SUBAPPLICATION Uebung_087a2_AX (* Beispiel für E_DEMUX_4, mit Plug and Socket *)
  (* Standard: 61499-2; Description: Copyright (c) 2026 Meisterschulen am Ostbahnhof This program and the accompanying materials are made available under the terms of the Eclipse Public License 2.0 which is available at https://www.eclipse.org/legal/epl-2.0/ SPDX-License-Identifier: EPL-2.0 *)
  (* Version 1.0, 2026-09-10, Franz Höpfinger, Meisterschulen am Ostbahnhof, initial API and implementation and/or initial documentation *)
  PACKAGE Uebungen;
  IMPORT logiBUS::io::DI::logiBUS_DI::Input_I1;
  IMPORT logiBUS::io::DI::logiBUS_DI::Input_I2;
  IMPORT logiBUS::io::DI::logiBUS_DI::Input_I3;
  IMPORT logiBUS::io::DI::logiBUS_DI::Input_I4;
  IMPORT logiBUS::io::DQ::logiBUS_DO::Output_Q1;
  IMPORT logiBUS::io::DQ::logiBUS_DO::Output_Q2;
  IMPORT logiBUS::io::DQ::logiBUS_DO::Output_Q3;
  IMPORT logiBUS::io::DQ::logiBUS_DO::Output_Q4;
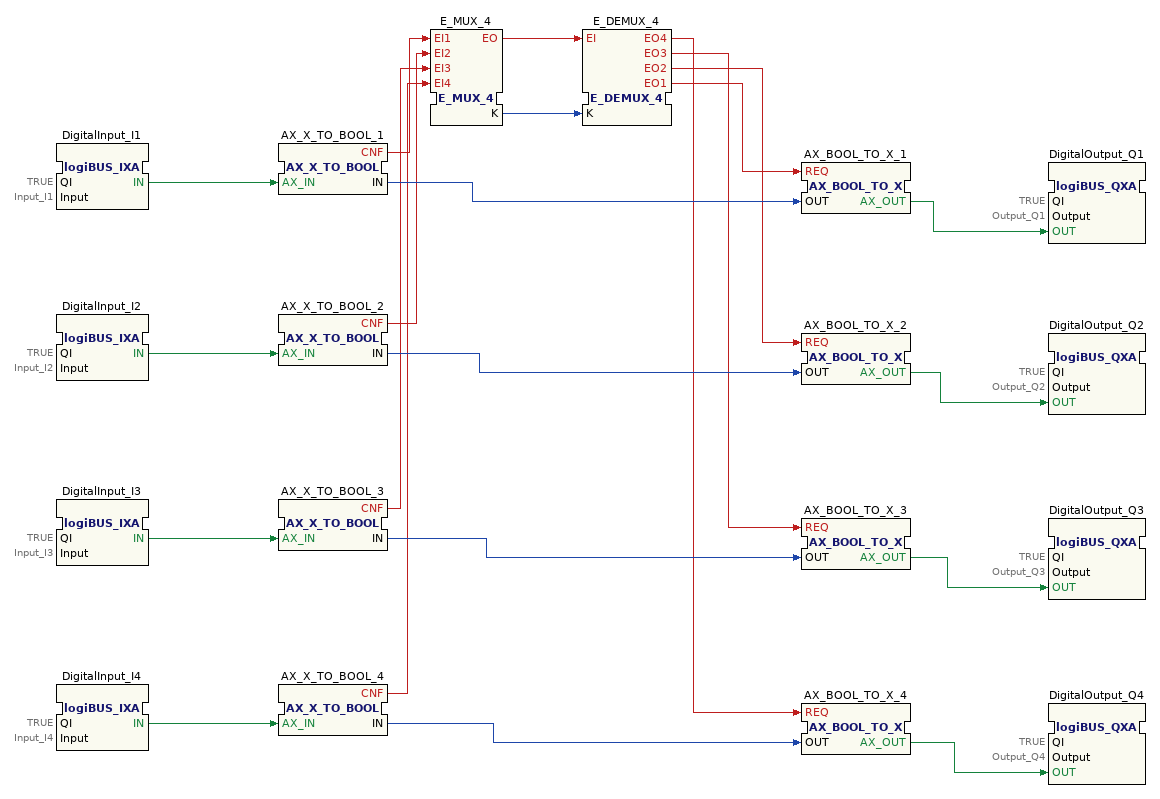
  FBS
    DigitalOutput_Q1 : logiBUS::io::DQ::logiBUS_QXA(QI := TRUE, Output := Output_Q1);
    DigitalInput_I1 : logiBUS::io::DI::logiBUS_IXA(QI := TRUE, Input := Input_I1);
    DigitalOutput_Q2 : logiBUS::io::DQ::logiBUS_QXA(QI := TRUE, Output := Output_Q2);
    DigitalInput_I2 : logiBUS::io::DI::logiBUS_IXA(QI := TRUE, Input := Input_I2);
    DigitalOutput_Q3 : logiBUS::io::DQ::logiBUS_QXA(QI := TRUE, Output := Output_Q3);
    DigitalInput_I3 : logiBUS::io::DI::logiBUS_IXA(QI := TRUE, Input := Input_I3);
    DigitalOutput_Q4 : logiBUS::io::DQ::logiBUS_QXA(QI := TRUE, Output := Output_Q4);
    DigitalInput_I4 : logiBUS::io::DI::logiBUS_IXA(QI := TRUE, Input := Input_I4);
    E_DEMUX_4 : iec61499::events::E_DEMUX_4;
    E_MUX_4 : iec61499::events::E_MUX_4;
    AX_X_TO_BOOL_1 : adapter::conversion::unidirectional::AX_X_TO_BOOL;
    AX_X_TO_BOOL_2 : adapter::conversion::unidirectional::AX_X_TO_BOOL;
    AX_X_TO_BOOL_3 : adapter::conversion::unidirectional::AX_X_TO_BOOL;
    AX_X_TO_BOOL_4 : adapter::conversion::unidirectional::AX_X_TO_BOOL;
    AX_BOOL_TO_X_1 : adapter::conversion::unidirectional::AX_BOOL_TO_X;
    AX_BOOL_TO_X_2 : adapter::conversion::unidirectional::AX_BOOL_TO_X;
    AX_BOOL_TO_X_3 : adapter::conversion::unidirectional::AX_BOOL_TO_X;
    AX_BOOL_TO_X_4 : adapter::conversion::unidirectional::AX_BOOL_TO_X;
  END_FBS
  EVENT_CONNECTIONS
    E_MUX_4.EO TO E_DEMUX_4.EI;
    AX_X_TO_BOOL_1.CNF TO E_MUX_4.EI1;
    AX_X_TO_BOOL_2.CNF TO E_MUX_4.EI2;
    AX_X_TO_BOOL_3.CNF TO E_MUX_4.EI3;
    AX_X_TO_BOOL_4.CNF TO E_MUX_4.EI4;
    E_DEMUX_4.EO4 TO AX_BOOL_TO_X_4.REQ;
    E_DEMUX_4.EO3 TO AX_BOOL_TO_X_3.REQ;
    E_DEMUX_4.EO2 TO AX_BOOL_TO_X_2.REQ;
    E_DEMUX_4.EO1 TO AX_BOOL_TO_X_1.REQ;
  END_CONNECTIONS
  DATA_CONNECTIONS
    E_MUX_4.K TO E_DEMUX_4.K;
    AX_X_TO_BOOL_1.IN TO AX_BOOL_TO_X_1.OUT;
    AX_X_TO_BOOL_2.IN TO AX_BOOL_TO_X_2.OUT;
    AX_X_TO_BOOL_3.IN TO AX_BOOL_TO_X_3.OUT;
    AX_X_TO_BOOL_4.IN TO AX_BOOL_TO_X_4.OUT;
  END_CONNECTIONS
  ADAPTER_CONNECTIONS
    DigitalInput_I1.IN TO AX_X_TO_BOOL_1.AX_IN;
    DigitalInput_I2.IN TO AX_X_TO_BOOL_2.AX_IN;
    DigitalInput_I3.IN TO AX_X_TO_BOOL_3.AX_IN;
    DigitalInput_I4.IN TO AX_X_TO_BOOL_4.AX_IN;
    AX_BOOL_TO_X_1.AX_OUT TO DigitalOutput_Q1.OUT;
    AX_BOOL_TO_X_2.AX_OUT TO DigitalOutput_Q2.OUT;
    AX_BOOL_TO_X_3.AX_OUT TO DigitalOutput_Q3.OUT;
    AX_BOOL_TO_X_4.AX_OUT TO DigitalOutput_Q4.OUT;
  END_CONNECTIONS
END_SUBAPPLICATION
